{attribute addProperty BoxType "EK1122-0000-0018"}
{attribute addProperty Id "Beckhoff_CXxxxxsub_EK1100EK1100_179A0949162A_0001_CX1100_0004_0000CX1100_179A0949162A_0003_CX1100_0004_0002CX1100_179A0949162A_0004_CX5010_EtherCAT_slaveCX5010_EtherCAT_slave_B56B2A0D16020A_0005_CX5010_EtherCAT_slaveCX5010_EtherCAT_slave_B56B2A0D16020A_0006_CX5020_EtherCAT_slaveCX5020_EtherCAT_slave_B56B2A0D16020A_0007_CX5020_EtherCAT_slaveCX5020_EtherCAT_slave_B56B2A0D16020A_0008_CX8010_EtherCAT_slaveCX8010_EtherCAT_slave_B56B2A0D16020A_0009_CX8010_EtherCAT_slaveCX8010_EtherCAT_slave_B56B2A0D16020A_0010_CX8110_EtherCAT_slaveCX8110_EtherCAT_slave_B56B2A0D16020A_0011_CX2020_EtherCAT_slaveCX2020_EtherCAT_slave_B56B2A0D16020A_0012_CX2020_EtherCAT_slaveCX2020_EtherCAT_slave_B56B2A0D16020A_0013_CX2020_EtherCAT_slaveCX2020_EtherCAT_slave_B56B2A0D16020A_0014_CX2030_EtherCAT_slaveCX2030_EtherCAT_slave_B56B2A0D16020A_0015_CX2030_EtherCAT_slaveCX2030_EtherCAT_slave_B56B2A0D16020A_0016_CX2030_EtherCAT_slaveCX2030_EtherCAT_slave_B56B2A0D16020A_0017_CX2033_EtherCAT_slaveCX2033_EtherCAT_slave_B56B2A0D16020A_0018_CX2040_EtherCAT_slaveCX2040_EtherCAT_slave_B56B2A0D16020A_0019_CX2040_EtherCAT_slaveCX2040_EtherCAT_slave_B56B2A0D16020A_0020_CX2040_EtherCAT_slaveCX2040_EtherCAT_slave_B56B2A0D16020A_0021_CX2042_EtherCAT_slaveCX2042_EtherCAT_slave_B56B2A0D16020A_0022_CX2043_EtherCAT_slaveCX2043_EtherCAT_slave_B56B2A0D16020A_0023_CX2062_EtherCAT_slaveCX2062_EtherCAT_slave_B56B2A0D16020A_0024_CX2072_EtherCAT_slaveCX2072_EtherCAT_slave_B56B2A0D16020A_0025_CX9020_EtherCAT_slaveCX9020_EtherCAT_slave_B56B2A0D16020A_0026_CX9020_EtherCAT_slaveCX9020_EtherCAT_slave_B56B2A0D16020A_0027_CX5120_EtherCAT_slaveCX5120_EtherCAT_slave_B56B2A0D16020A_0028_CX5130_EtherCAT_slaveCX5130_EtherCAT_slave_B56B2A0D16020A_0029_CX5140_EtherCAT_slaveCX5140_EtherCAT_slave_B56B2A0D16020A_0030_CX5230_EtherCAT_slaveCX5230_EtherCAT_slave_B56B2A0D16020A_0031_CX5240_EtherCAT_slaveCX5240_EtherCAT_slave_B56B2A0D16020A_0002_CX1100_0004_0001CX1100_179A0949162"}
{attribute addProperty CRC "1943729630"}
{attribute addProperty SizeInBites "4544"}
{attribute addProperty SizeInBytes "568"}
TYPE Beckhoff_CXxxxxEK1122_73DAF5DE EXTENDS EK1122_179A0949 :
STRUCT
	{attribute addProperty Name "Beckhoff_CXxxxxsub_EK1100"}
	Beckhoff_CXxxxxsub_EK1100 : EK1100_179A0949;
	{attribute addProperty Name "A_0001_CX1100_0004_0000"}
	A_0001_CX1100_0004_0000 : CX1100_179A0949;
	{attribute addProperty Name "A_0003_CX1100_0004_0002"}
	A_0003_CX1100_0004_0002 : CX1100_179A0949;
	{attribute addProperty Name "A_0004_CX5010_EtherCAT_slave"}
	A_0004_CX5010_EtherCAT_slave : CX5010_EtherCAT_slave_B56B2A0D;
	{attribute addProperty Name "A_0005_CX5010_EtherCAT_slave"}
	A_0005_CX5010_EtherCAT_slave : CX5010_EtherCAT_slave_B56B2A0D;
	{attribute addProperty Name "A_0006_CX5020_EtherCAT_slave"}
	A_0006_CX5020_EtherCAT_slave : CX5020_EtherCAT_slave_B56B2A0D;
	{attribute addProperty Name "A_0007_CX5020_EtherCAT_slave"}
	A_0007_CX5020_EtherCAT_slave : CX5020_EtherCAT_slave_B56B2A0D;
	{attribute addProperty Name "A_0008_CX8010_EtherCAT_slave"}
	A_0008_CX8010_EtherCAT_slave : CX8010_EtherCAT_slave_B56B2A0D;
	{attribute addProperty Name "A_0009_CX8010_EtherCAT_slave"}
	A_0009_CX8010_EtherCAT_slave : CX8010_EtherCAT_slave_B56B2A0D;
	{attribute addProperty Name "A_0010_CX8110_EtherCAT_slave"}
	A_0010_CX8110_EtherCAT_slave : CX8110_EtherCAT_slave_B56B2A0D;
	{attribute addProperty Name "A_0011_CX2020_EtherCAT_slave"}
	A_0011_CX2020_EtherCAT_slave : CX2020_EtherCAT_slave_B56B2A0D;
	{attribute addProperty Name "A_0012_CX2020_EtherCAT_slave"}
	A_0012_CX2020_EtherCAT_slave : CX2020_EtherCAT_slave_B56B2A0D;
	{attribute addProperty Name "A_0013_CX2020_EtherCAT_slave"}
	A_0013_CX2020_EtherCAT_slave : CX2020_EtherCAT_slave_B56B2A0D;
	{attribute addProperty Name "A_0014_CX2030_EtherCAT_slave"}
	A_0014_CX2030_EtherCAT_slave : CX2030_EtherCAT_slave_B56B2A0D;
	{attribute addProperty Name "A_0015_CX2030_EtherCAT_slave"}
	A_0015_CX2030_EtherCAT_slave : CX2030_EtherCAT_slave_B56B2A0D;
	{attribute addProperty Name "A_0016_CX2030_EtherCAT_slave"}
	A_0016_CX2030_EtherCAT_slave : CX2030_EtherCAT_slave_B56B2A0D;
	{attribute addProperty Name "A_0017_CX2033_EtherCAT_slave"}
	A_0017_CX2033_EtherCAT_slave : CX2033_EtherCAT_slave_B56B2A0D;
	{attribute addProperty Name "A_0018_CX2040_EtherCAT_slave"}
	A_0018_CX2040_EtherCAT_slave : CX2040_EtherCAT_slave_B56B2A0D;
	{attribute addProperty Name "A_0019_CX2040_EtherCAT_slave"}
	A_0019_CX2040_EtherCAT_slave : CX2040_EtherCAT_slave_B56B2A0D;
	{attribute addProperty Name "A_0020_CX2040_EtherCAT_slave"}
	A_0020_CX2040_EtherCAT_slave : CX2040_EtherCAT_slave_B56B2A0D;
	{attribute addProperty Name "A_0021_CX2042_EtherCAT_slave"}
	A_0021_CX2042_EtherCAT_slave : CX2042_EtherCAT_slave_B56B2A0D;
	{attribute addProperty Name "A_0022_CX2043_EtherCAT_slave"}
	A_0022_CX2043_EtherCAT_slave : CX2043_EtherCAT_slave_B56B2A0D;
	{attribute addProperty Name "A_0023_CX2062_EtherCAT_slave"}
	A_0023_CX2062_EtherCAT_slave : CX2062_EtherCAT_slave_B56B2A0D;
	{attribute addProperty Name "A_0024_CX2072_EtherCAT_slave"}
	A_0024_CX2072_EtherCAT_slave : CX2072_EtherCAT_slave_B56B2A0D;
	{attribute addProperty Name "A_0025_CX9020_EtherCAT_slave"}
	A_0025_CX9020_EtherCAT_slave : CX9020_EtherCAT_slave_B56B2A0D;
	{attribute addProperty Name "A_0026_CX9020_EtherCAT_slave"}
	A_0026_CX9020_EtherCAT_slave : CX9020_EtherCAT_slave_B56B2A0D;
	{attribute addProperty Name "A_0027_CX5120_EtherCAT_slave"}
	A_0027_CX5120_EtherCAT_slave : CX5120_EtherCAT_slave_B56B2A0D;
	{attribute addProperty Name "A_0028_CX5130_EtherCAT_slave"}
	A_0028_CX5130_EtherCAT_slave : CX5130_EtherCAT_slave_B56B2A0D;
	{attribute addProperty Name "A_0029_CX5140_EtherCAT_slave"}
	A_0029_CX5140_EtherCAT_slave : CX5140_EtherCAT_slave_B56B2A0D;
	{attribute addProperty Name "A_0030_CX5230_EtherCAT_slave"}
	A_0030_CX5230_EtherCAT_slave : CX5230_EtherCAT_slave_B56B2A0D;
	{attribute addProperty Name "A_0031_CX5240_EtherCAT_slave"}
	A_0031_CX5240_EtherCAT_slave : CX5240_EtherCAT_slave_B56B2A0D;
	{attribute addProperty Name "A_0002_CX1100_0004_0001"}
	A_0002_CX1100_0004_0001 : CX1100_179A0949;
END_STRUCT
END_TYPE

(* stored: Version 1.2.0.0, ProductVersion 3.1.4024.9
   DUT Beckhoff_CXxxxxEK1122_73DAF5DE: Id {55016b1d-04b5-400a-ad02-72dfb5bebca5} *)
